{attribute 'qualified_only'}
{attribute 'strict'}
{attribute 'to_string'}
TYPE TurtleNames :
(
	Batman := 1,Superman:=2
);
END_TYPE

(* stored: Version 1.1.0.1
   DUT TurtleNames: Id {babf16e0-1567-4563-878f-d7bb7aba76d1} *)
